// TIA Portal V16 export
// export: Created 2023-01-03T15:35:07.7120292Z, ExportSetting WithDefaults, DisplayName Totally Integrated Automation Portal, DisplayVersion V16, DisplayName TIA Portal Version Control Interface, DisplayVersion V16, DisplayName TIA Portal Openness, DisplayVersion V16, DisplayName STEP 7 Professional, DisplayVersion V16, DisplayName STEP 7 Safety, DisplayVersion V16, DisplayName WinCC Advanced, DisplayVersion V16
FUNCTION "MOTOR_SPEEDMONITORING" : Void   // FC3, LAD
{ S7_Optimized_Access := 'TRUE' }
VERSION : 0.1
// stored: AutoNumber true, IsIECCheckEnabled false, SetENOAutomatically false, UDAEnableTagReadback false
   VAR_INPUT
      Act_speed_val : Int;
   END_VAR
   VAR_OUTPUT
      fault_detected : Bool;
   END_VAR
   VAR_IN_OUT
      motor_speed_in_rpm : Int;
      err_speed_max_fw : Bool;
      warning_speed_max_fw : Bool;
      warning_speed_min_reverse : Bool;
      err_speed_min_reverse : Bool;
   END_VAR
   VAR_TEMP
      out2 : Real;
   END_VAR
BEGIN

REGION Network 1
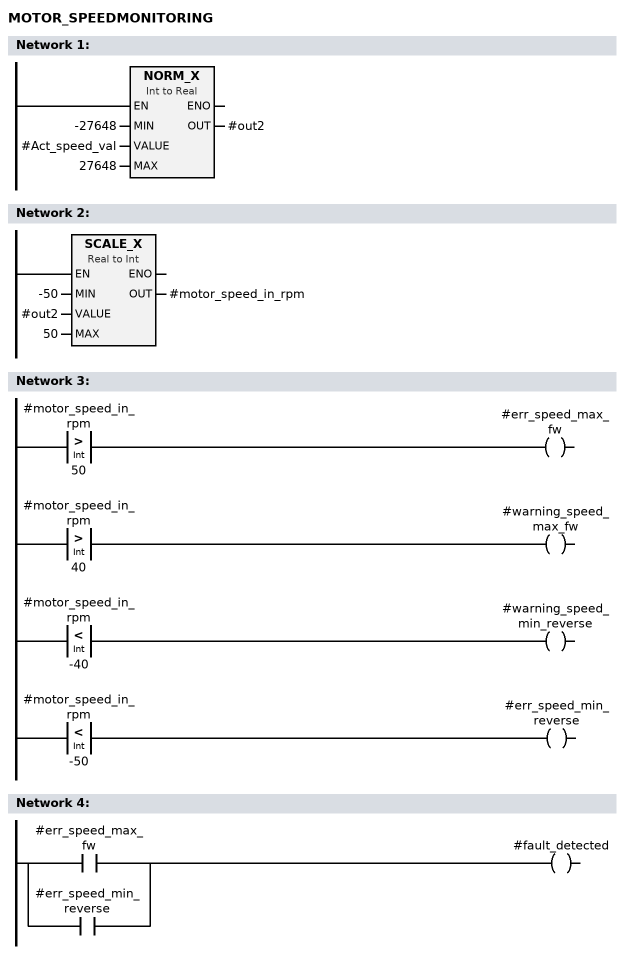
   RUNG wire#powerrail
      { S7_Templates := "[SrcType := Int, DestType := Real]" } Normalize(min := -27648, value := #Act_speed_val, max := 27648, out => #out2)
   END_RUNG
   // the same network as SCL:
   #out2 := NORM_X(MIN := -27648, VALUE := #Act_speed_val, MAX := 27648);
END_REGION

REGION Network 2
   RUNG wire#powerrail
      { S7_Templates := "[SrcType := Real, DestType := Int]" } Scale(min := -50, value := #out2, max := 50, out => #motor_speed_in_rpm)
   END_RUNG
   // the same network as SCL:
   #motor_speed_in_rpm := SCALE_X(MIN := -50, VALUE := #out2, MAX := 50);
END_REGION

REGION Network 3
   RUNG wire#powerrail
      { S7_Templates := "SrcType := Int" } GT_Contact(in1 := #motor_speed_in_rpm, in2 := 50)
      Coil( #err_speed_max_fw )
   END_RUNG
   RUNG wire#powerrail
      { S7_Templates := "SrcType := Int" } GT_Contact(in1 := #motor_speed_in_rpm, in2 := 40)
      Coil( #warning_speed_max_fw )
   END_RUNG
   RUNG wire#powerrail
      { S7_Templates := "SrcType := Int" } LT_Contact(in1 := #motor_speed_in_rpm, in2 := -40)
      Coil( #warning_speed_min_reverse )
   END_RUNG
   RUNG wire#powerrail
      { S7_Templates := "SrcType := Int" } LT_Contact(in1 := #motor_speed_in_rpm, in2 := -50)
      Coil( #err_speed_min_reverse )
   END_RUNG
   // the same network as SCL:
   #err_speed_max_fw := #motor_speed_in_rpm > 50;
   #warning_speed_max_fw := #motor_speed_in_rpm > 40;
   #warning_speed_min_reverse := #motor_speed_in_rpm < (-40);
   #err_speed_min_reverse := #motor_speed_in_rpm < (-50);
END_REGION

REGION Network 4
   RUNG wire#powerrail
      Contact( #err_speed_max_fw )
      wire#w1
      Coil( #fault_detected )
   END_RUNG
   RUNG wire#powerrail
      Contact( #err_speed_min_reverse )
   END_RUNG wire#w1
   // the same network as SCL:
   #fault_detected := #err_speed_max_fw OR #err_speed_min_reverse;
END_REGION
END_FUNCTION
